# EPICS substitutions: epics/db/EL6695.substitutions
file "./db/ecSlave.template"
{
  pattern {}
          {}
}

# No custom data yet
#file "./db/EL6695.template"
#{
#  pattern {}
#          {}
#}
